// Mitsubishi GX Works2 project: 十字路口交通灯控制   PLC: FX1S

PROGRAM MAIN
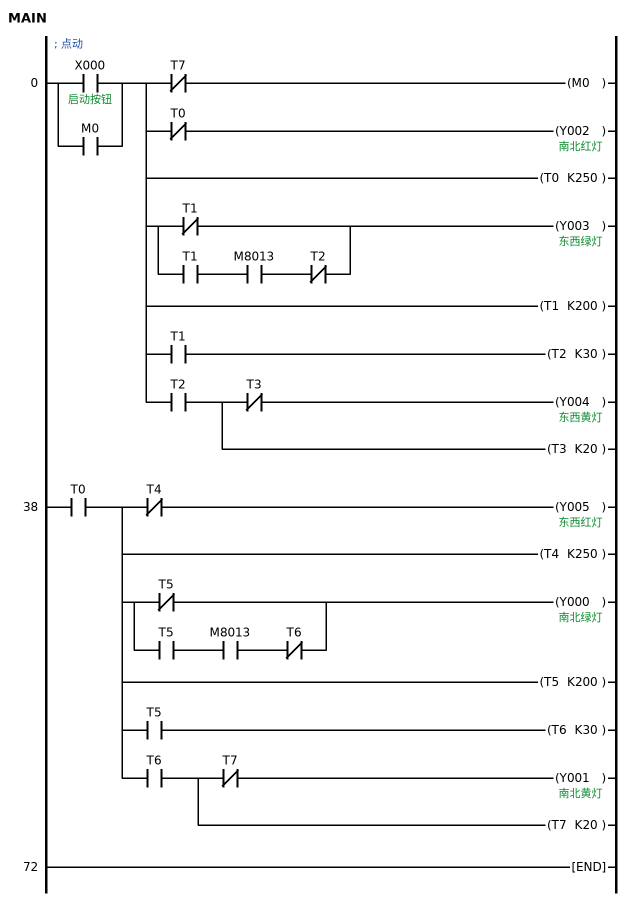
; 点动
0     LD      X000  ; 启动按钮
      OR      M0
      MPS
      ANI     T7
      OUT     M0
      MRD
      ANI     T0
      OUT     Y002  ; 南北红灯
      MPP
      OUT     T0 K250
      MPS
      LDI     T1
      LD      T1
      AND     M8013
      ANI     T2
      ORB
      ANB
      OUT     Y003  ; 东西绿灯
      MPP
      OUT     T1 K200
      MPS
      AND     T1
      OUT     T2 K30
      MPP
      AND     T2
      MPS
      ANI     T3
      OUT     Y004  ; 东西黄灯
      MPP
      OUT     T3 K20
38    LD      T0
      MPS
      ANI     T4
      OUT     Y005  ; 东西红灯
      MPP
      OUT     T4 K250
      MPS
      LDI     T5
      LD      T5
      AND     M8013
      ANI     T6
      ORB
      ANB
      OUT     Y000  ; 南北绿灯
      MPP
      OUT     T5 K200
      MPS
      AND     T5
      OUT     T6 K30
      MPP
      AND     T6
      MPS
      ANI     T7
      OUT     Y001  ; 南北黄灯
      MPP
      OUT     T7 K20
72    END
END_PROGRAM
